{attribute addProperty BoxType "EP4174-0002-0016"}
{attribute addProperty Id "AO_Outputs_ChannelAT %Q*ARRAY[0..3] OF AO_Outputs_Channel_F57FA4F96480WcStateAT %I*WcState_64F6A8C6810InfoDataAT %I*InfoData_BC63D37F80100"}
{attribute addProperty CRC "645842055"}
{attribute addProperty SizeInBites "152"}
{attribute addProperty SizeInBytes "19"}
TYPE EP4174_253CF8AE :
STRUCT
	{attribute addProperty Name "AO_Outputs_Channel"}
	AO_Outputs_Channel : ARRAY[0..3] OF AO_Outputs_Channel_F57FA4F9;
	{attribute addProperty Name "WcState"}
	WcState : WcState_64F6A8C6;
	{attribute addProperty Name "InfoData"}
	InfoData : InfoData_BC63D37F;
END_STRUCT
END_TYPE

(* stored: Version 1.2.0.0, ProductVersion 3.1.4024.9
   DUT EP4174_253CF8AE: Id {d8f479d0-f600-4d88-88f3-342bff27469b} *)
